// TIA Portal V16 export
// export: Created 2024-09-05T17:39:17.4210446Z, ExportSetting WithDefaults, DisplayName Totally Integrated Automation Portal, DisplayVersion V16 Update 6, DisplayName TIA Portal Version Control Interface, DisplayVersion V16 Update 2, DisplayName TIA Portal Openness, DisplayVersion V16 Update 6, DisplayName STEP 7 Professional, DisplayVersion V16 Update 6, DisplayName STEP 7 Safety, DisplayVersion V16, DisplayName WinCC Advanced, DisplayVersion V16 Update 6
DATA_BLOCK "DB_ProductionCountersEdit"   // DB66
{ S7_Optimized_Access := 'TRUE' }
VERSION : 0.1
// stored: AutoNumber true, DBAccessibleFromOPCUA true, IsOnlyStoredInLoadMemory false, IsRetainMemResEnabled false, IsWriteProtectedInAS false, MemoryReserve 100
   VAR
      ProgramNumber : Int := 1;
      ProgramName : String[50] := '2569703X-LH';
      ProductCounters { S7_SetPoint := 'True'} : "UDT_ProductionProgramCounters";
      SettingsCanBeChanged : Bool := FALSE;
      DeleteCounters : Int := 0;
   END_VAR
BEGIN
   ProductCounters.Product[1].Shift[1..3].Ok := 0;
   ProductCounters.Product[2].Shift[1..3].Ok := 0;
   ProductCounters.Product[3].Shift[1..3].Ok := 0;
   ProductCounters.Product[4].Shift[1..3].Ok := 0;
   ProductCounters.Product[5].Shift[1..3].Ok := 0;
   ProductCounters.Product[6].Shift[1..3].Ok := 0;
   ProductCounters.Product[7].Shift[1..3].Ok := 0;
   ProductCounters.Product[8].Shift[1..3].Ok := 0;
   ProductCounters.Product[1].Shift[1..3].Nok := 0;
   ProductCounters.Product[2].Shift[1..3].Nok := 0;
   ProductCounters.Product[3].Shift[1..3].Nok := 0;
   ProductCounters.Product[4].Shift[1..3].Nok := 0;
   ProductCounters.Product[5].Shift[1..3].Nok := 0;
   ProductCounters.Product[6].Shift[1..3].Nok := 0;
   ProductCounters.Product[7].Shift[1..3].Nok := 0;
   ProductCounters.Product[8].Shift[1..3].Nok := 0;
   ProductCounters.Product[1..8].Overall.Ok := 0;
   ProductCounters.Product[1..8].Overall.Nok := 0;
END_DATA_BLOCK
